FUNCTION_BLOCK FB_Ventilation EXTENDS FB_ActuatorContinous
VAR_INPUT
END_VAR
VAR_OUTPUT
END_VAR
VAR
END_VAR

END_FUNCTION_BLOCK

(* stored: Version 1.1.0.1, ProductVersion 3.1.4024.10
   POU FB_Ventilation: Id {b3736a55-8dec-49ad-8b80-0e1e5782a762}, SpecialFunc None *)
